TYPE ST_DebugColumnBIO :
STRUCT

//<DIO>
	ipDBColumnPCWLeakage				: E_BackdoorState;
	ipDBColumnPCWSupplyLeakage    		: E_BackdoorState;
	ipDBColumnPCWReturnLeakage    		: E_BackdoorState;
	                                    
	opDBColumnHotAirExhaustFan 			:BOOL;
	opDBColumnPCWValve         			:BOOL;
	opDBColumnTstAirSol        			:BOOL;
	opDBColumnAPAirSol         			:BOOL;
//</DIO>

//<CVTIO>
	ipDBColumnPCWRegularFlowSensor		:REAL;
	ipDBColumnPCWSupplyPressure       	:REAL;
	ipDBColumnPCWReturnPressure       	:REAL;
	ipDBColumnTstAirPressure          	:REAL;
	ipDBColumnAPAirPressure           	:REAL;
	ipDBColumnDewPointSensor          	:REAL;
	ipDBColumnTempSensor 	:REAL;
	ipDBColumnPCWSupplyTemperature    	:REAL;
	ipDBColumnPCWReturnTemperature    	:REAL;
//</CVTIO>

END_STRUCT
END_TYPE

(* stored: Version 1.1.0.1, ProductVersion 3.1.4022.18
   DUT ST_DebugColumnBIO: Id {0da78fb2-0c87-4d27-8163-efefe3836047} *)
